	//HORA COMPLETA
	IF 	LA_IHM.HORARIO_ATUAL_SEGUNDO = 59 	AND
		LA_IHM.HORARIO_ATUAL_MINUTO  = 59	THEN
		LA_IHM.bit_HORARIO_HORA_COMPLETO	:=	TRUE;
	ELSE
		LA_IHM.bit_HORARIO_HORA_COMPLETO	:=	FALSE;
	END_IF
	
	//DIA COMPLETO
	IF 	LA_IHM.HORARIO_ATUAL_SEGUNDO = 57 	AND
		LA_IHM.HORARIO_ATUAL_MINUTO  = 59	AND
		LA_IHM.HORARIO_ATUAL_HORA	  = 5	OR
		teste_dia						 	THEN
		LA_IHM.bit_HORARIO_DIA_COMPLETO	:=	TRUE;
	ELSE
		LA_IHM.bit_HORARIO_DIA_COMPLETO	:=	FALSE;
	END_IF
	
	//DIA REAL COMPLETO
	IF 	LA_IHM.HORARIO_ATUAL_SEGUNDO = 58 	AND
		LA_IHM.HORARIO_ATUAL_MINUTO  = 59	AND
		LA_IHM.HORARIO_ATUAL_HORA	  = 23	THEN
		LA_IHM.bit_HORARIO_DIA_COMPLETO_REAL	:=	TRUE;
	ELSE
		LA_IHM.bit_HORARIO_DIA_COMPLETO_REAL	:=	FALSE;
	END_IF

//TIMER RETENTIVOS TURNO MAQUINA RODANDO
pvar.RTON_tmr_MAQUINA_RODANDO_T1(T_IN:= LA_IHM.turno_A AND LA_GERAL.bit_STATUS_RODANDO, T_PT:= T#999999999MS);
pvar.RTON_tmr_MAQUINA_RODANDO_T2(T_IN:= LA_IHM.turno_B AND LA_GERAL.bit_STATUS_RODANDO, T_PT:= T#999999999MS);
pvar.RTON_tmr_MAQUINA_RODANDO_T3(T_IN:= LA_IHM.turno_C AND LA_GERAL.bit_STATUS_RODANDO, T_PT:= T#999999999MS);

//TIMER RETENTIVOS TURNO MAQUINA PARADA
pvar.RTON_tmr_MAQUINA_PARADA_T1(T_IN:= LA_IHM.turno_A AND LA_GERAL.bit_STATUS_PARADA, T_PT:= T#999999999MS);
pvar.RTON_tmr_MAQUINA_PARADA_T2(T_IN:= LA_IHM.turno_B AND LA_GERAL.bit_STATUS_PARADA, T_PT:= T#999999999MS);
pvar.RTON_tmr_MAQUINA_PARADA_T3(T_IN:= LA_IHM.turno_C AND LA_GERAL.bit_STATUS_PARADA, T_PT:= T#999999999MS);

//TIMER RETENTIVOS TURNO MAQUINA OCIOSA
pvar.RTON_tmr_MAQUINA_OCIOSA_T1(T_IN:= LA_IHM.turno_A AND LA_GERAL.bit_STATUS_OCIOSA, T_PT:= T#999999999MS);
pvar.RTON_tmr_MAQUINA_OCIOSA_T2(T_IN:= LA_IHM.turno_B AND LA_GERAL.bit_STATUS_OCIOSA, T_PT:= T#999999999MS);
pvar.RTON_tmr_MAQUINA_OCIOSA_T3(T_IN:= LA_IHM.turno_C AND LA_GERAL.bit_STATUS_OCIOSA, T_PT:= T#999999999MS);

//================================================================================================================================================================================
//================================================================================================================================================================================

//--------//--------//-------//------CONTADORES------//--------------//-----------//-----------//------------//


//CONTAGEM PILHAS PESADAS OK TURNO A
pvar.cont_PILHAS_COMPLETADAS_TURNO_1(
	CU:= GVL_PESAGEM.bit_PESAGEM_ATUAL AND (LA_GERAL.bit_STATUS_RODANDO OR LA_GERAL.bit_STATUS_OCIOSA) AND LA_IHM.turno_A);
	
//CONTAGEM PILHAS PESADAS OK TURNO B
pvar.cont_PILHAS_COMPLETADAS_TURNO_2(
	CU:= GVL_PESAGEM.bit_PESAGEM_ATUAL AND (LA_GERAL.bit_STATUS_RODANDO OR LA_GERAL.bit_STATUS_OCIOSA) AND LA_IHM.turno_B);
	
//CONTAGEM PILHAS PESADAS OK TURNO C
pvar.cont_PILHAS_COMPLETADAS_TURNO_3(
	CU:= GVL_PESAGEM.bit_PESAGEM_ATUAL AND (LA_GERAL.bit_STATUS_RODANDO OR LA_GERAL.bit_STATUS_OCIOSA) AND LA_IHM.turno_C);

//CONTAGEM PILHAS REJEITADAS TURNO A
pvar.cont_PILHAS_REJEITADAS_TURNO_1(
	CU:= GVL_PESAGEM.bit_PESAGEM_ERRO AND (LA_GERAL.bit_STATUS_RODANDO OR LA_GERAL.bit_STATUS_OCIOSA) AND LA_IHM.turno_A);
	
//CONTAGEM PILHAS REJEITADAS TURNO B
pvar.cont_PILHAS_REJEITADAS_TURNO_2(
	CU:= GVL_PESAGEM.bit_PESAGEM_ERRO AND (LA_GERAL.bit_STATUS_RODANDO OR LA_GERAL.bit_STATUS_OCIOSA) AND LA_IHM.turno_B);
	
//CONTAGEM PILHAS REJEITADAS TURNO C
pvar.cont_PILHAS_REJEITADAS_TURNO_3(
	CU:= GVL_PESAGEM.bit_PESAGEM_ERRO AND (LA_GERAL.bit_STATUS_RODANDO OR LA_GERAL.bit_STATUS_OCIOSA) AND LA_IHM.turno_C);
	
//CONTAGEM PILHAS TOTAL TURNO A
pvar.cont_PILHAS_TOTAL_TURNO_1(
	CU:= (GVL_PESAGEM.bit_PESAGEM_ATUAL OR GVL_PESAGEM.bit_PESAGEM_ERRO) AND (LA_GERAL.bit_STATUS_RODANDO OR LA_GERAL.bit_STATUS_OCIOSA OR teste) AND LA_IHM.turno_A);
	
//CONTAGEM PILHAS TOTAL TURNO B
pvar.cont_PILHAS_TOTAL_TURNO_2(
	CU:= (GVL_PESAGEM.bit_PESAGEM_ATUAL OR GVL_PESAGEM.bit_PESAGEM_ERRO) AND (LA_GERAL.bit_STATUS_RODANDO OR LA_GERAL.bit_STATUS_OCIOSA) AND LA_IHM.turno_B);
	
//CONTAGEM PILHAS TOTAL TURNO C
pvar.cont_PILHAS_TOTAL_TURNO_3(
	CU:= (GVL_PESAGEM.bit_PESAGEM_ATUAL OR GVL_PESAGEM.bit_PESAGEM_ERRO) AND (LA_GERAL.bit_STATUS_RODANDO OR LA_GERAL.bit_STATUS_OCIOSA) AND LA_IHM.turno_C);
	
//--------//--------//-------//------EFICIENCIA------//--------------//-----------//-----------//------------//
//garante que não haverá erros de divisão por 0. A eficiencia só é contada a partir de quando a contagem POR TEMPO começou
	
//PORCENTAGEM DE PILHAS COMPLETADAS TURNO 1
IF PVAR.ihm_PILHAS_TOTAL_TURNO_ARRAY.PRIMEIRO[0] > 0 THEN
	LA_IHM.num_PORCENTAGEM_COMPLETADAS_T1	:=	(DINT_TO_REAL(PVAR.ihm_PILHAS_COMPLETADAS_TURNO_ARRAY.PRIMEIRO[0]) / DINT_TO_REAL(PVAR.ihm_PILHAS_TOTAL_TURNO_ARRAY.PRIMEIRO[0])) * 100;
END_IF

//PORCENTAGEM DE PILHAS COMPLETADAS TURNO 2
IF PVAR.ihm_PILHAS_TOTAL_TURNO_ARRAY.SEGUNDO[0] > 0 THEN
	LA_IHM.num_PORCENTAGEM_COMPLETADAS_T2	:=	(DINT_TO_REAL(PVAR.ihm_PILHAS_COMPLETADAS_TURNO_ARRAY.SEGUNDO[0]) / DINT_TO_REAL(PVAR.ihm_PILHAS_TOTAL_TURNO_ARRAY.SEGUNDO[0])) * 100;
END_IF

//PORCENTAGEM DE PILHAS COMPLETADAS TURNO 3
IF PVAR.ihm_PILHAS_TOTAL_TURNO_ARRAY.TERCEIRO[0] > 0 THEN
	LA_IHM.num_PORCENTAGEM_COMPLETADAS_T3	:=	(DINT_TO_REAL(PVAR.ihm_PILHAS_COMPLETADAS_TURNO_ARRAY.TERCEIRO[0]) / DINT_TO_REAL(PVAR.ihm_PILHAS_TOTAL_TURNO_ARRAY.TERCEIRO[0])) * 100;
END_IF


//PORCENTAGEM DE PILHAS REJEITADAS TURNO 1
IF PVAR.ihm_PILHAS_TOTAL_TURNO_ARRAY.PRIMEIRO[0] > 0 THEN
	LA_IHM.num_PORCENTAGEM_REJEITADAS_T1	:=	100 - LA_IHM.num_PORCENTAGEM_COMPLETADAS_T1;
END_IF

//PORCENTAGEM DE PILHAS REJEITADAS TURNO 2
IF PVAR.ihm_PILHAS_TOTAL_TURNO_ARRAY.SEGUNDO[0] > 0 THEN
	LA_IHM.num_PORCENTAGEM_REJEITADAS_T2	:=	100 - LA_IHM.num_PORCENTAGEM_COMPLETADAS_T2;
END_IF

//PORCENTAGEM DE PILHAS REJEITADAS TURNO 3
IF PVAR.ihm_PILHAS_TOTAL_TURNO_ARRAY.TERCEIRO[0] > 0 THEN
	LA_IHM.num_PORCENTAGEM_REJEITADAS_T3	:=	100 - LA_IHM.num_PORCENTAGEM_COMPLETADAS_T3;
END_IF


//================================================================================================================================================================================
//================================================================================================================================================================================
//RESET DE VARIÁVEIS NA TROCA DE TURNO

	IF tmr_TURNO_TROCADO.Q THEN
		pvar.RTON_tmr_MAQUINA_RODANDO_T1.Timer_reset	:=	TRUE;
		pvar.RTON_tmr_MAQUINA_RODANDO_T2.Timer_reset	:=	TRUE;
		pvar.RTON_tmr_MAQUINA_RODANDO_T3.Timer_reset	:=	TRUE;
		
		pvar.RTON_tmr_MAQUINA_PARADA_T1.Timer_reset	:=	TRUE;
		pvar.RTON_tmr_MAQUINA_PARADA_T2.Timer_reset	:=	TRUE;
		pvar.RTON_tmr_MAQUINA_PARADA_T3.Timer_reset	:=	TRUE;
		
		pvar.RTON_tmr_MAQUINA_OCIOSA_T1.Timer_reset	:=	TRUE;
		pvar.RTON_tmr_MAQUINA_OCIOSA_T2.Timer_reset	:=	TRUE;
		pvar.RTON_tmr_MAQUINA_OCIOSA_T3.Timer_reset	:=	TRUE;
		
		PVAR.cont_PILHAS_COMPLETADAS_TURNO_1.RESET	:=	TRUE;
		PVAR.cont_PILHAS_COMPLETADAS_TURNO_2.RESET	:=	TRUE;
		PVAR.cont_PILHAS_COMPLETADAS_TURNO_3.RESET	:=	TRUE;
		
		PVAR.cont_PILHAS_REJEITADAS_TURNO_1.RESET	:=	TRUE;
		PVAR.cont_PILHAS_REJEITADAS_TURNO_2.RESET	:=	TRUE;
		PVAR.cont_PILHAS_REJEITADAS_TURNO_3.RESET	:=	TRUE;
		
		PVAR.cont_PILHAS_TOTAL_TURNO_1.RESET		:=	TRUE;
		PVAR.cont_PILHAS_TOTAL_TURNO_2.RESET		:=	TRUE;
		PVAR.cont_PILHAS_TOTAL_TURNO_3.RESET		:=	TRUE;
		
		LA_GERAL.bit_TURNO_TROCADO				:= FALSE;
	ELSE
		pvar.RTON_tmr_MAQUINA_RODANDO_T1.Timer_reset	:=	FALSE;
		pvar.RTON_tmr_MAQUINA_RODANDO_T2.Timer_reset	:=	FALSE;
		pvar.RTON_tmr_MAQUINA_RODANDO_T3.Timer_reset	:=	FALSE;
		
		pvar.RTON_tmr_MAQUINA_PARADA_T1.Timer_reset	:=	FALSE;
		pvar.RTON_tmr_MAQUINA_PARADA_T2.Timer_reset	:=	FALSE;
		pvar.RTON_tmr_MAQUINA_PARADA_T3.Timer_reset	:=	FALSE;
		
		pvar.RTON_tmr_MAQUINA_OCIOSA_T1.Timer_reset	:=	FALSE;
		pvar.RTON_tmr_MAQUINA_OCIOSA_T2.Timer_reset	:=	FALSE;
		pvar.RTON_tmr_MAQUINA_OCIOSA_T3.Timer_reset	:=	FALSE;
		
		PVAR.cont_PILHAS_COMPLETADAS_TURNO_1.RESET	:=	FALSE;
		PVAR.cont_PILHAS_COMPLETADAS_TURNO_2.RESET	:=	FALSE;
		PVAR.cont_PILHAS_COMPLETADAS_TURNO_3.RESET	:=	FALSE;
		
		PVAR.cont_PILHAS_REJEITADAS_TURNO_1.RESET	:=	FALSE;
		PVAR.cont_PILHAS_REJEITADAS_TURNO_2.RESET	:=	FALSE;
		PVAR.cont_PILHAS_REJEITADAS_TURNO_3.RESET	:=	FALSE;
		
		PVAR.cont_PILHAS_TOTAL_TURNO_1.RESET		:=	FALSE;
		PVAR.cont_PILHAS_TOTAL_TURNO_2.RESET		:=	FALSE;
		PVAR.cont_PILHAS_TOTAL_TURNO_3.RESET		:=	FALSE;
		
	END_IF
	
//RESETAR MANUALMENTE CONTADORES DO TURNO A
	IF LA_IHM.bit_CONTADORES_RESET	AND LA_IHM.turno_A THEN
		pvar.RTON_tmr_MAQUINA_RODANDO_T1.Timer_reset	:=	TRUE;
		pvar.RTON_tmr_MAQUINA_PARADA_T1.Timer_reset		:=	TRUE;
		pvar.RTON_tmr_MAQUINA_OCIOSA_T1.Timer_reset		:=	TRUE;
		PVAR.cont_PILHAS_COMPLETADAS_TURNO_1.RESET		:=	TRUE;
		PVAR.cont_PILHAS_REJEITADAS_TURNO_1.RESET		:=	TRUE;
		PVAR.cont_PILHAS_TOTAL_TURNO_1.RESET			:=	TRUE;
	END_IF
	
//RESETAR MANUALMENTE CONTADORES DO TURNO B
	IF LA_IHM.bit_CONTADORES_RESET	AND LA_IHM.turno_B THEN
		pvar.RTON_tmr_MAQUINA_RODANDO_T2.Timer_reset	:=	TRUE;
		pvar.RTON_tmr_MAQUINA_PARADA_T2.Timer_reset		:=	TRUE;
		pvar.RTON_tmr_MAQUINA_OCIOSA_T2.Timer_reset		:=	TRUE;
		PVAR.cont_PILHAS_COMPLETADAS_TURNO_2.RESET		:=	TRUE;
		PVAR.cont_PILHAS_REJEITADAS_TURNO_2.RESET		:=	TRUE;
		PVAR.cont_PILHAS_TOTAL_TURNO_2.RESET			:=	TRUE;
	END_IF
	
//RESETAR MANUALMENTE CONTADORES DO TURNO C
	IF LA_IHM.bit_CONTADORES_RESET	AND LA_IHM.turno_C THEN
		pvar.RTON_tmr_MAQUINA_RODANDO_T3.Timer_reset	:=	TRUE;
		pvar.RTON_tmr_MAQUINA_PARADA_T3.Timer_reset		:=	TRUE;
		pvar.RTON_tmr_MAQUINA_OCIOSA_T3.Timer_reset		:=	TRUE;
		PVAR.cont_PILHAS_COMPLETADAS_TURNO_3.RESET		:=	TRUE;
		PVAR.cont_PILHAS_REJEITADAS_TURNO_3.RESET		:=	TRUE;
		PVAR.cont_PILHAS_TOTAL_TURNO_3.RESET			:=	TRUE;
	END_IF


//RESETAR CONTADORES DOS TURNOS 05:59:55
	IF 	(LA_IHM.HORARIO_ATUAL_HORA 	 = 5	AND
		LA_IHM.HORARIO_ATUAL_MINUTO = 59		AND
		LA_IHM.HORARIO_ATUAL_SEGUNDO = 55)		OR
		teste_reset_cont_turnoa					THEN
			LA_GERAL.bit_TURNO_TROCADO	:= TRUE;
	END_IF

tmr_TURNO_TROCADO		(IN := LA_GERAL.bit_TURNO_TROCADO,  PT := T#4S);


//LIMITE DE HORÁRIOS DOS TURNOS
LIM_HORA_TURNO1(IN:= LA_IHM.HORARIO_ATUAL_HORA, HIGH:= 13, LOW:= 6);
LIM_HORA_TURNO2(IN:= LA_IHM.HORARIO_ATUAL_HORA, HIGH:= 21, LOW:= 14);
LIM_HORA_TURNO3(IN:= LA_IHM.HORARIO_ATUAL_HORA, HIGH:= 5, LOW:= 22);

E06_HISTORICO();
E07_HISTORICO_ESPELHAMENTO();

END_PROGRAM

// LADO_A/05 - LA_IHM/E06_HISTORICO
PROGRAM E06_HISTORICO
VAR
	HORARIO_ATUAL_DIA_ANTERIOR	: DINT;
END_VAR

	IF LA_IHM.bit_HORARIO_DIA_COMPLETO_REAL THEN
		LA_IHM.info_DIA_ANTERIOR := LA_IHM.HORARIO_ATUAL_DIA;
		LA_IHM.info_MES_ANTERIOR := LA_IHM.HORARIO_ATUAL_MES;
	END_IF
	
//================================================================================================================================================================================
//================================================================================================================================================================================
//ARMAZENAMENTO DE DADOS DE PRODUÇÃO DE TURNO

	//ARMAZENAMENTO DE DADOS DE PRODUÇÃO TURNO A
	IF LA_IHM.turno_A	THEN
		
		PVAR.IHM_DIA_TURNO_ARRAY.PRIMEIRO[0] := LA_IHM.HORARIO_ATUAL_DIA;
		PVAR.IHM_MES_TURNO_ARRAY.PRIMEIRO[0] := LA_IHM.HORARIO_ATUAL_MES;
		
		PVAR.IHM_TEMPO_RODANDO_ARRAY.PRIMEIRO[0] := TIME_TO_DINT(pvar.RTON_tmr_MAQUINA_RODANDO_T1.RTON_ET);
		PVAR.IHM_TEMPO_PARADO_ARRAY.PRIMEIRO[0]  := TIME_TO_DINT(pvar.RTON_tmr_MAQUINA_PARADA_T1.RTON_ET);
		PVAR.IHM_TEMPO_OCIOSO_ARRAY.PRIMEIRO[0]  := TIME_TO_DINT(pvar.RTON_tmr_MAQUINA_OCIOSA_T1.RTON_ET);
	
		PVAR.ihm_PILHAS_COMPLETADAS_TURNO_ARRAY.PRIMEIRO[0]		:=	pvar.cont_PILHAS_COMPLETADAS_TURNO_1.CV;
		PVAR.ihm_PILHAS_REJEITADAS_TURNO_ARRAY.PRIMEIRO[0]		:=	pvar.cont_PILHAS_REJEITADAS_TURNO_1.CV;
		PVAR.ihm_PILHAS_TOTAL_TURNO_ARRAY.PRIMEIRO[0]			:=	pvar.cont_PILHAS_TOTAL_TURNO_1.CV;
		
		PVAR.ihm_PILHAS_COMPLETADAS_PORCENTAGEM_TURNO_ARRAY.PRIMEIRO[0]	:=	REAL_TO_DINT(LA_IHM.num_PORCENTAGEM_COMPLETADAS_T1);
		PVAR.ihm_PILHAS_REJEITADAS_PORCENTAGEM_TURNO_ARRAY.PRIMEIRO[0]	:=	REAL_TO_DINT(LA_IHM.num_PORCENTAGEM_REJEITADAS_T1);
	END_IF
	
	//ARMAZENAMENTO DE DADOS DE PRODUÇÃO TURNO B
	IF LA_IHM.turno_B	THEN
		
		PVAR.IHM_DIA_TURNO_ARRAY.SEGUNDO[0] := LA_IHM.HORARIO_ATUAL_DIA;
		PVAR.IHM_MES_TURNO_ARRAY.SEGUNDO[0] := LA_IHM.HORARIO_ATUAL_MES;
		
		PVAR.IHM_TEMPO_RODANDO_ARRAY.SEGUNDO[0] := TIME_TO_DINT(pvar.RTON_tmr_MAQUINA_RODANDO_T2.RTON_ET);
		PVAR.IHM_TEMPO_PARADO_ARRAY.SEGUNDO[0]  := TIME_TO_DINT(pvar.RTON_tmr_MAQUINA_PARADA_T2.RTON_ET);
		PVAR.IHM_TEMPO_OCIOSO_ARRAY.SEGUNDO[0]  := TIME_TO_DINT(pvar.RTON_tmr_MAQUINA_OCIOSA_T2.RTON_ET);
		
		PVAR.ihm_PILHAS_COMPLETADAS_TURNO_ARRAY.SEGUNDO[0]		:=	pvar.cont_PILHAS_COMPLETADAS_TURNO_2.CV;
		PVAR.ihm_PILHAS_REJEITADAS_TURNO_ARRAY.SEGUNDO[0]		:=	pvar.cont_PILHAS_REJEITADAS_TURNO_2.CV;
		PVAR.ihm_PILHAS_TOTAL_TURNO_ARRAY.SEGUNDO[0]			:=	pvar.cont_PILHAS_TOTAL_TURNO_2.CV;
		
		PVAR.ihm_PILHAS_COMPLETADAS_PORCENTAGEM_TURNO_ARRAY.SEGUNDO[0]	:=	REAL_TO_DINT(LA_IHM.num_PORCENTAGEM_COMPLETADAS_T2);
		PVAR.ihm_PILHAS_REJEITADAS_PORCENTAGEM_TURNO_ARRAY.SEGUNDO[0]	:=	REAL_TO_DINT(LA_IHM.num_PORCENTAGEM_REJEITADAS_T2);
	END_IF
	
	//ARMAZENAMENTO DE DADOS DE PRODUÇÃO TURNO C
	IF LA_IHM.turno_C	THEN
	
	IF LA_IHM.HORARIO_ATUAL_HORA <= 5 THEN
		PVAR.IHM_DIA_TURNO_ARRAY.TERCEIRO[0] := LA_IHM.HORARIO_ATUAL_DIA - 1;
		PVAR.IHM_MES_TURNO_ARRAY.TERCEIRO[0] := LA_IHM.HORARIO_ATUAL_MES;
	ELSE
		PVAR.IHM_DIA_TURNO_ARRAY.TERCEIRO[0] := LA_IHM.HORARIO_ATUAL_DIA;
		PVAR.IHM_MES_TURNO_ARRAY.TERCEIRO[0] := LA_IHM.HORARIO_ATUAL_MES;
	END_IF
		
		PVAR.IHM_TEMPO_RODANDO_ARRAY.TERCEIRO[0] := TIME_TO_DINT(pvar.RTON_tmr_MAQUINA_RODANDO_T3.RTON_ET);
		PVAR.IHM_TEMPO_PARADO_ARRAY.TERCEIRO[0]  := TIME_TO_DINT(pvar.RTON_tmr_MAQUINA_PARADA_T3.RTON_ET);
		PVAR.IHM_TEMPO_OCIOSO_ARRAY.TERCEIRO[0]  := TIME_TO_DINT(pvar.RTON_tmr_MAQUINA_OCIOSA_T3.RTON_ET);
		
		PVAR.ihm_PILHAS_COMPLETADAS_TURNO_ARRAY.TERCEIRO[0]		:=	pvar.cont_PILHAS_COMPLETADAS_TURNO_3.CV;
		PVAR.ihm_PILHAS_REJEITADAS_TURNO_ARRAY.TERCEIRO[0]		:=	pvar.cont_PILHAS_REJEITADAS_TURNO_3.CV;
		PVAR.ihm_PILHAS_TOTAL_TURNO_ARRAY.TERCEIRO[0]			:=	pvar.cont_PILHAS_TOTAL_TURNO_3.CV;
		
		PVAR.ihm_PILHAS_COMPLETADAS_PORCENTAGEM_TURNO_ARRAY.TERCEIRO[0]	:=	REAL_TO_DINT(LA_IHM.num_PORCENTAGEM_COMPLETADAS_T3);
		PVAR.ihm_PILHAS_REJEITADAS_PORCENTAGEM_TURNO_ARRAY.TERCEIRO[0]	:=	REAL_TO_DINT(LA_IHM.num_PORCENTAGEM_REJEITADAS_T3);
	END_IF
	
	
//================================================================================================================================================================================
//================================================================================================================================================================================
//SHIFT NO ARMAZENAMENTO DE DADOS DE PRODUÇÃO DE TURNO

//---------------//---------------DIA COMPLETO PRIMEIRO---------------//---------------//---------------//---------------//---------------//---------------//---------------//---------------//---------------//---------------//---------------//---------------//
	LA_IHM.COP_ihm_DIA_TURNO(Source:= ADR(PVAR.IHM_DIA_TURNO_ARRAY.PRIMEIRO[0]) , Dest:= ADR(PVAR.IHM_DIA_TURNO_ARRAY_AUX.PRIMEIRO[0]), Length:= 10, Trigger:= LA_IHM.bit_HORARIO_DIA_COMPLETO);
	LA_IHM.COP_ihm_DIA_TURNO_AUX(Source:= ADR(PVAR.IHM_DIA_TURNO_ARRAY_AUX.PRIMEIRO[0]) , Dest:= ADR(PVAR.IHM_DIA_TURNO_ARRAY.PRIMEIRO[1]), Length:= 9, Trigger:= LA_IHM.bit_HORARIO_DIA_COMPLETO);
	
	LA_IHM.COP_ihm_MES_TURNO(Source:= ADR(PVAR.IHM_MES_TURNO_ARRAY.PRIMEIRO[0]) , Dest:= ADR(PVAR.IHM_MES_TURNO_ARRAY_AUX.PRIMEIRO[0]), Length:= 10, Trigger:= LA_IHM.bit_HORARIO_DIA_COMPLETO);
	LA_IHM.COP_ihm_MES_TURNO_AUX(Source:= ADR(PVAR.IHM_MES_TURNO_ARRAY_AUX.PRIMEIRO[0]) , Dest:= ADR(PVAR.IHM_MES_TURNO_ARRAY.PRIMEIRO[1]), Length:= 9, Trigger:= LA_IHM.bit_HORARIO_DIA_COMPLETO);
	
	LA_IHM.COP_ihm_RODANDO_TURNO(Source:= ADR(PVAR.IHM_TEMPO_RODANDO_ARRAY.PRIMEIRO[0]) , Dest:= ADR(PVAR.IHM_TEMPO_RODANDO_ARRAY_AUX.PRIMEIRO[0]), Length:= 10, Trigger:= LA_IHM.bit_HORARIO_DIA_COMPLETO);
	LA_IHM.COP_ihm_RODANDO_TURNO_AUX(Source:= ADR(PVAR.IHM_TEMPO_RODANDO_ARRAY_AUX.PRIMEIRO[0]) , Dest:= ADR(PVAR.IHM_TEMPO_RODANDO_ARRAY.PRIMEIRO[1]), Length:= 9, Trigger:= LA_IHM.bit_HORARIO_DIA_COMPLETO);
	
	LA_IHM.COP_ihm_PARADO_TURNO(Source:= ADR(PVAR.IHM_TEMPO_PARADO_ARRAY.PRIMEIRO[0]) , Dest:= ADR(PVAR.IHM_TEMPO_PARADO_ARRAY_AUX.PRIMEIRO[0]), Length:= 10, Trigger:= LA_IHM.bit_HORARIO_DIA_COMPLETO);
	LA_IHM.COP_ihm_PARADO_TURNO_AUX(Source:= ADR(PVAR.IHM_TEMPO_PARADO_ARRAY_AUX.PRIMEIRO[0]) , Dest:= ADR(PVAR.IHM_TEMPO_PARADO_ARRAY.PRIMEIRO[1]), Length:= 9, Trigger:= LA_IHM.bit_HORARIO_DIA_COMPLETO);
	
	LA_IHM.COP_ihm_OCIOSO_TURNO(Source:= ADR(PVAR.IHM_TEMPO_OCIOSO_ARRAY.PRIMEIRO[0]) , Dest:= ADR(PVAR.IHM_TEMPO_OCIOSO_ARRAY_AUX.PRIMEIRO[0]), Length:= 10, Trigger:= LA_IHM.bit_HORARIO_DIA_COMPLETO);
	LA_IHM.COP_ihm_OCIOSO_TURNO_AUX(Source:= ADR(PVAR.IHM_TEMPO_OCIOSO_ARRAY_AUX.PRIMEIRO[0]) , Dest:= ADR(PVAR.IHM_TEMPO_OCIOSO_ARRAY.PRIMEIRO[1]), Length:= 9, Trigger:= LA_IHM.bit_HORARIO_DIA_COMPLETO);
		
	LA_IHM.COP_ihm_PILHAS_COMPLETADAS_TURNO(Source:= ADR(PVAR.ihm_PILHAS_COMPLETADAS_TURNO_ARRAY.PRIMEIRO[0]) , Dest:= ADR(PVAR.ihm_PILHAS_COMPLETADAS_TURNO_ARRAY_AUX.PRIMEIRO[0]), Length:= 10, Trigger:= LA_IHM.bit_HORARIO_DIA_COMPLETO);
	LA_IHM.COP_ihm_PILHAS_COMPLETADAS_TURNO_AUX(Source:= ADR(PVAR.ihm_PILHAS_COMPLETADAS_TURNO_ARRAY_AUX.PRIMEIRO[0]) , Dest:= ADR(PVAR.ihm_PILHAS_COMPLETADAS_TURNO_ARRAY.PRIMEIRO[1]), Length:= 9, Trigger:= LA_IHM.bit_HORARIO_DIA_COMPLETO);
	
	LA_IHM.COP_ihm_PILHAS_REJEITADAS_TURNO(Source:= ADR(PVAR.ihm_PILHAS_REJEITADAS_TURNO_ARRAY.PRIMEIRO[0]) , Dest:= ADR(PVAR.ihm_PILHAS_REJEITADAS_TURNO_ARRAY_AUX.PRIMEIRO[0]), Length:= 10, Trigger:= LA_IHM.bit_HORARIO_DIA_COMPLETO);
	LA_IHM.COP_ihm_PILHAS_REJEITADAS_TURNO_AUX(Source:= ADR(PVAR.ihm_PILHAS_REJEITADAS_TURNO_ARRAY_AUX.PRIMEIRO[0]) , Dest:= ADR(PVAR.ihm_PILHAS_REJEITADAS_TURNO_ARRAY.PRIMEIRO[1]), Length:= 9, Trigger:= LA_IHM.bit_HORARIO_DIA_COMPLETO);
	
	LA_IHM.COP_ihm_PILHAS_TOTAL_TURNO(Source:= ADR(PVAR.ihm_PILHAS_TOTAL_TURNO_ARRAY.PRIMEIRO[0]) , Dest:= ADR(PVAR.ihm_PILHAS_TOTAL_TURNO_ARRAY_AUX.PRIMEIRO[0]), Length:= 10, Trigger:= LA_IHM.bit_HORARIO_DIA_COMPLETO);
	LA_IHM.COP_ihm_PILHAS_TOTAL_TURNO_AUX(Source:= ADR(PVAR.ihm_PILHAS_TOTAL_TURNO_ARRAY_AUX.PRIMEIRO[0]) , Dest:= ADR(PVAR.ihm_PILHAS_TOTAL_TURNO_ARRAY.PRIMEIRO[1]), Length:= 9, Trigger:= LA_IHM.bit_HORARIO_DIA_COMPLETO);
	
	LA_IHM.COP_ihm_PORCENTAGEM_COMPLETADAS(Source:= ADR(PVAR.ihm_PILHAS_COMPLETADAS_PORCENTAGEM_TURNO_ARRAY.PRIMEIRO[0]) , Dest:= ADR(PVAR.ihm_PILHAS_COMPLETADAS_PORCENTAGEM_TURNO_ARRAY_AUX.PRIMEIRO[0]), Length:= 10, Trigger:= LA_IHM.bit_HORARIO_DIA_COMPLETO);
	LA_IHM.COP_ihm_PORCENTAGEM_COMPLETADAS_AUX(Source:= ADR(PVAR.ihm_PILHAS_COMPLETADAS_PORCENTAGEM_TURNO_ARRAY_AUX.PRIMEIRO[0]) , Dest:= ADR(PVAR.ihm_PILHAS_COMPLETADAS_PORCENTAGEM_TURNO_ARRAY.PRIMEIRO[1]), Length:= 9, Trigger:= LA_IHM.bit_HORARIO_DIA_COMPLETO);
	
	LA_IHM.COP_ihm_PORCENTAGEM_REJEITADAS(Source:= ADR(PVAR.ihm_PILHAS_REJEITADAS_PORCENTAGEM_TURNO_ARRAY.PRIMEIRO[0]) , Dest:= ADR(PVAR.ihm_PILHAS_REJEITADAS_PORCENTAGEM_TURNO_ARRAY_AUX.PRIMEIRO[0]), Length:= 10, Trigger:= LA_IHM.bit_HORARIO_DIA_COMPLETO);
	LA_IHM.COP_ihm_PORCENTAGEM_REJEITADAS_AUX(Source:= ADR(PVAR.ihm_PILHAS_REJEITADAS_PORCENTAGEM_TURNO_ARRAY_AUX.PRIMEIRO[0]) , Dest:= ADR(PVAR.ihm_PILHAS_REJEITADAS_PORCENTAGEM_TURNO_ARRAY.PRIMEIRO[1]), Length:= 9, Trigger:= LA_IHM.bit_HORARIO_DIA_COMPLETO);
	
//---------------//---------------//---------------//---------------//---------------//---------------//---------------//---------------//---------------//---------------//---------------//---------------//---------------//---------------//---------------//---------------//	
//---------------//---------------//---------------//---------------//---------------//---------------//---------------//---------------//---------------//---------------//---------------//---------------//---------------//---------------//---------------//---------------//
//---------------//---------------DIA COMPLETO SEGUNDO---------------//---------------//---------------//---------------//---------------//---------------//---------------//---------------//---------------//---------------//---------------//---------------//
	LA_IHM.COP_ihm_DIA_TURNO2(Source:= ADR(PVAR.IHM_DIA_TURNO_ARRAY.SEGUNDO[0]) , Dest:= ADR(PVAR.IHM_DIA_TURNO_ARRAY_AUX.SEGUNDO[0]), Length:= 10, Trigger:= LA_IHM.bit_HORARIO_DIA_COMPLETO);
	LA_IHM.COP_ihm_DIA_TURNO_AUX2(Source:= ADR(PVAR.IHM_DIA_TURNO_ARRAY_AUX.SEGUNDO[0]) , Dest:= ADR(PVAR.IHM_DIA_TURNO_ARRAY.SEGUNDO[1]), Length:= 9, Trigger:= LA_IHM.bit_HORARIO_DIA_COMPLETO);
	
	LA_IHM.COP_ihm_MES_TURNO2(Source:= ADR(PVAR.IHM_MES_TURNO_ARRAY.SEGUNDO[0]) , Dest:= ADR(PVAR.IHM_MES_TURNO_ARRAY_AUX.SEGUNDO[0]), Length:= 10, Trigger:= LA_IHM.bit_HORARIO_DIA_COMPLETO);
	LA_IHM.COP_ihm_MES_TURNO_AUX2(Source:= ADR(PVAR.IHM_MES_TURNO_ARRAY_AUX.SEGUNDO[0]) , Dest:= ADR(PVAR.IHM_MES_TURNO_ARRAY.SEGUNDO[1]), Length:= 9, Trigger:= LA_IHM.bit_HORARIO_DIA_COMPLETO);

	LA_IHM.COP_ihm_RODANDO_TURNO2(Source:= ADR(PVAR.IHM_TEMPO_RODANDO_ARRAY.SEGUNDO[0]) , Dest:= ADR(PVAR.IHM_TEMPO_RODANDO_ARRAY_AUX.SEGUNDO[0]), Length:= 10, Trigger:= LA_IHM.bit_HORARIO_DIA_COMPLETO);
	LA_IHM.COP_ihm_RODANDO_TURNO_AUX2(Source:= ADR(PVAR.IHM_TEMPO_RODANDO_ARRAY_AUX.SEGUNDO[0]) , Dest:= ADR(PVAR.IHM_TEMPO_RODANDO_ARRAY.SEGUNDO[1]), Length:= 9, Trigger:= LA_IHM.bit_HORARIO_DIA_COMPLETO);
	
	LA_IHM.COP_ihm_PARADO_TURNO2(Source:= ADR(PVAR.IHM_TEMPO_PARADO_ARRAY.SEGUNDO[0]) , Dest:= ADR(PVAR.IHM_TEMPO_PARADO_ARRAY_AUX.SEGUNDO[0]), Length:= 10, Trigger:= LA_IHM.bit_HORARIO_DIA_COMPLETO);
	LA_IHM.COP_ihm_PARADO_TURNO_AUX2(Source:= ADR(PVAR.IHM_TEMPO_PARADO_ARRAY_AUX.SEGUNDO[0]) , Dest:= ADR(PVAR.IHM_TEMPO_PARADO_ARRAY.SEGUNDO[1]), Length:= 9, Trigger:= LA_IHM.bit_HORARIO_DIA_COMPLETO);
	
	LA_IHM.COP_ihm_OCIOSO_TURNO2(Source:= ADR(PVAR.IHM_TEMPO_OCIOSO_ARRAY.SEGUNDO[0]) , Dest:= ADR(PVAR.IHM_TEMPO_OCIOSO_ARRAY_AUX.SEGUNDO[0]), Length:= 10, Trigger:= LA_IHM.bit_HORARIO_DIA_COMPLETO);
	LA_IHM.COP_ihm_OCIOSO_TURNO_AUX2(Source:= ADR(PVAR.IHM_TEMPO_OCIOSO_ARRAY_AUX.SEGUNDO[0]) , Dest:= ADR(PVAR.IHM_TEMPO_OCIOSO_ARRAY.SEGUNDO[1]), Length:= 9, Trigger:= LA_IHM.bit_HORARIO_DIA_COMPLETO);
	
	LA_IHM.COP_ihm_PILHAS_COMPLETADAS_TURNO2(Source:= ADR(PVAR.ihm_PILHAS_COMPLETADAS_TURNO_ARRAY.SEGUNDO[0]) , Dest:= ADR(PVAR.ihm_PILHAS_COMPLETADAS_TURNO_ARRAY_AUX.SEGUNDO[0]), Length:= 10, Trigger:= LA_IHM.bit_HORARIO_DIA_COMPLETO);
	LA_IHM.COP_ihm_PILHAS_COMPLETADAS_TURNO_AUX2(Source:= ADR(PVAR.ihm_PILHAS_COMPLETADAS_TURNO_ARRAY_AUX.SEGUNDO[0]) , Dest:= ADR(PVAR.ihm_PILHAS_COMPLETADAS_TURNO_ARRAY.SEGUNDO[1]), Length:= 9, Trigger:= LA_IHM.bit_HORARIO_DIA_COMPLETO);
	
	LA_IHM.COP_ihm_PILHAS_REJEITADAS_TURNO2(Source:= ADR(PVAR.ihm_PILHAS_REJEITADAS_TURNO_ARRAY.SEGUNDO[0]) , Dest:= ADR(PVAR.ihm_PILHAS_REJEITADAS_TURNO_ARRAY_AUX.SEGUNDO[0]), Length:= 10, Trigger:= LA_IHM.bit_HORARIO_DIA_COMPLETO);
	LA_IHM.COP_ihm_PILHAS_REJEITADAS_TURNO_AUX2(Source:= ADR(PVAR.ihm_PILHAS_REJEITADAS_TURNO_ARRAY_AUX.SEGUNDO[0]) , Dest:= ADR(PVAR.ihm_PILHAS_REJEITADAS_TURNO_ARRAY.SEGUNDO[1]), Length:= 9, Trigger:= LA_IHM.bit_HORARIO_DIA_COMPLETO);
	
	LA_IHM.COP_ihm_PILHAS_TOTAL_TURNO2(Source:= ADR(PVAR.ihm_PILHAS_TOTAL_TURNO_ARRAY.SEGUNDO[0]) , Dest:= ADR(PVAR.ihm_PILHAS_TOTAL_TURNO_ARRAY_AUX.SEGUNDO[0]), Length:= 10, Trigger:= LA_IHM.bit_HORARIO_DIA_COMPLETO);
	LA_IHM.COP_ihm_PILHAS_TOTAL_TURNO_AUX2(Source:= ADR(PVAR.ihm_PILHAS_TOTAL_TURNO_ARRAY_AUX.SEGUNDO[0]) , Dest:= ADR(PVAR.ihm_PILHAS_TOTAL_TURNO_ARRAY.SEGUNDO[1]), Length:= 9, Trigger:= LA_IHM.bit_HORARIO_DIA_COMPLETO);
	
	LA_IHM.COP_ihm_PORCENTAGEM_COMPLETADAS2(Source:= ADR(PVAR.ihm_PILHAS_COMPLETADAS_PORCENTAGEM_TURNO_ARRAY.SEGUNDO[0]) , Dest:= ADR(PVAR.ihm_PILHAS_COMPLETADAS_PORCENTAGEM_TURNO_ARRAY_AUX.SEGUNDO[0]), Length:= 10, Trigger:= LA_IHM.bit_HORARIO_DIA_COMPLETO);
	LA_IHM.COP_ihm_PORCENTAGEM_COMPLETADAS_AUX2(Source:= ADR(PVAR.ihm_PILHAS_COMPLETADAS_PORCENTAGEM_TURNO_ARRAY_AUX.SEGUNDO[0]) , Dest:= ADR(PVAR.ihm_PILHAS_COMPLETADAS_PORCENTAGEM_TURNO_ARRAY.SEGUNDO[1]), Length:= 9, Trigger:= LA_IHM.bit_HORARIO_DIA_COMPLETO);
	
	LA_IHM.COP_ihm_PORCENTAGEM_REJEITADAS2(Source:= ADR(PVAR.ihm_PILHAS_REJEITADAS_PORCENTAGEM_TURNO_ARRAY.SEGUNDO[0]) , Dest:= ADR(PVAR.ihm_PILHAS_REJEITADAS_PORCENTAGEM_TURNO_ARRAY_AUX.SEGUNDO[0]), Length:= 10, Trigger:= LA_IHM.bit_HORARIO_DIA_COMPLETO);
	LA_IHM.COP_ihm_PORCENTAGEM_REJEITADAS_AUX2(Source:= ADR(PVAR.ihm_PILHAS_REJEITADAS_PORCENTAGEM_TURNO_ARRAY_AUX.SEGUNDO[0]) , Dest:= ADR(PVAR.ihm_PILHAS_REJEITADAS_PORCENTAGEM_TURNO_ARRAY.SEGUNDO[1]), Length:= 9, Trigger:= LA_IHM.bit_HORARIO_DIA_COMPLETO);
//---------------//---------------//---------------//---------------//---------------//---------------//---------------//---------------//---------------//---------------//---------------//---------------//---------------//---------------//---------------//---------------//	
//---------------//---------------//---------------//---------------//---------------//---------------//---------------//---------------//---------------//---------------//---------------//---------------//---------------//---------------//---------------//---------------//
//---------------//---------------DIA COMPLETO TERCEIRO---------------//---------------//---------------//---------------//---------------//---------------//---------------//---------------//---------------//---------------//---------------//---------------//
	LA_IHM.COP_ihm_DIA_TURNO3(Source:= ADR(PVAR.IHM_DIA_TURNO_ARRAY.TERCEIRO[0]) , Dest:= ADR(PVAR.IHM_DIA_TURNO_ARRAY_AUX.TERCEIRO[0]), Length:= 10, Trigger:= LA_IHM.bit_HORARIO_DIA_COMPLETO);
	LA_IHM.COP_ihm_DIA_TURNO_AUX3(Source:= ADR(PVAR.IHM_DIA_TURNO_ARRAY_AUX.TERCEIRO[0]) , Dest:= ADR(PVAR.IHM_DIA_TURNO_ARRAY.TERCEIRO[1]), Length:= 9, Trigger:= LA_IHM.bit_HORARIO_DIA_COMPLETO);
	
	LA_IHM.COP_ihm_MES_TURNO3(Source:= ADR(PVAR.IHM_MES_TURNO_ARRAY.TERCEIRO[0]) , Dest:= ADR(PVAR.IHM_MES_TURNO_ARRAY_AUX.TERCEIRO[0]), Length:= 10, Trigger:= LA_IHM.bit_HORARIO_DIA_COMPLETO);
	LA_IHM.COP_ihm_MES_TURNO_AUX3(Source:= ADR(PVAR.IHM_MES_TURNO_ARRAY_AUX.TERCEIRO[0]) , Dest:= ADR(PVAR.IHM_MES_TURNO_ARRAY.TERCEIRO[1]), Length:= 9, Trigger:= LA_IHM.bit_HORARIO_DIA_COMPLETO);

	LA_IHM.COP_ihm_RODANDO_TURNO3(Source:= ADR(PVAR.IHM_TEMPO_RODANDO_ARRAY.TERCEIRO[0]) , Dest:= ADR(PVAR.IHM_TEMPO_RODANDO_ARRAY_AUX.TERCEIRO[0]), Length:= 10, Trigger:= LA_IHM.bit_HORARIO_DIA_COMPLETO);
	LA_IHM.COP_ihm_RODANDO_TURNO_AUX3(Source:= ADR(PVAR.IHM_TEMPO_RODANDO_ARRAY_AUX.TERCEIRO[0]) , Dest:= ADR(PVAR.IHM_TEMPO_RODANDO_ARRAY.TERCEIRO[1]), Length:= 9, Trigger:= LA_IHM.bit_HORARIO_DIA_COMPLETO);
	
	LA_IHM.COP_ihm_PARADO_TURNO3(Source:= ADR(PVAR.IHM_TEMPO_PARADO_ARRAY.TERCEIRO[0]) , Dest:= ADR(PVAR.IHM_TEMPO_PARADO_ARRAY_AUX.TERCEIRO[0]), Length:= 10, Trigger:= LA_IHM.bit_HORARIO_DIA_COMPLETO);
	LA_IHM.COP_ihm_PARADO_TURNO_AUX3(Source:= ADR(PVAR.IHM_TEMPO_PARADO_ARRAY_AUX.TERCEIRO[0]) , Dest:= ADR(PVAR.IHM_TEMPO_PARADO_ARRAY.TERCEIRO[1]), Length:= 9, Trigger:= LA_IHM.bit_HORARIO_DIA_COMPLETO);
	
	LA_IHM.COP_ihm_OCIOSO_TURNO3(Source:= ADR(PVAR.IHM_TEMPO_OCIOSO_ARRAY.TERCEIRO[0]) , Dest:= ADR(PVAR.IHM_TEMPO_OCIOSO_ARRAY_AUX.TERCEIRO[0]), Length:= 10, Trigger:= LA_IHM.bit_HORARIO_DIA_COMPLETO);
	LA_IHM.COP_ihm_OCIOSO_TURNO_AUX3(Source:= ADR(PVAR.IHM_TEMPO_OCIOSO_ARRAY_AUX.TERCEIRO[0]) , Dest:= ADR(PVAR.IHM_TEMPO_OCIOSO_ARRAY.TERCEIRO[1]), Length:= 9, Trigger:= LA_IHM.bit_HORARIO_DIA_COMPLETO);
	
	LA_IHM.COP_ihm_PILHAS_COMPLETADAS_TURNO3(Source:= ADR(PVAR.ihm_PILHAS_COMPLETADAS_TURNO_ARRAY.TERCEIRO[0]) , Dest:= ADR(PVAR.ihm_PILHAS_COMPLETADAS_TURNO_ARRAY_AUX.TERCEIRO[0]), Length:= 10, Trigger:= LA_IHM.bit_HORARIO_DIA_COMPLETO);
	LA_IHM.COP_ihm_PILHAS_COMPLETADAS_TURNO_AUX3(Source:= ADR(PVAR.ihm_PILHAS_COMPLETADAS_TURNO_ARRAY_AUX.TERCEIRO[0]) , Dest:= ADR(PVAR.ihm_PILHAS_COMPLETADAS_TURNO_ARRAY.TERCEIRO[1]), Length:= 9, Trigger:= LA_IHM.bit_HORARIO_DIA_COMPLETO);
	
	LA_IHM.COP_ihm_PILHAS_REJEITADAS_TURNO3(Source:= ADR(PVAR.ihm_PILHAS_REJEITADAS_TURNO_ARRAY.TERCEIRO[0]) , Dest:= ADR(PVAR.ihm_PILHAS_REJEITADAS_TURNO_ARRAY_AUX.TERCEIRO[0]), Length:= 10, Trigger:= LA_IHM.bit_HORARIO_DIA_COMPLETO);
	LA_IHM.COP_ihm_PILHAS_REJEITADAS_TURNO_AUX3(Source:= ADR(PVAR.ihm_PILHAS_REJEITADAS_TURNO_ARRAY_AUX.TERCEIRO[0]) , Dest:= ADR(PVAR.ihm_PILHAS_REJEITADAS_TURNO_ARRAY.TERCEIRO[1]), Length:= 9, Trigger:= LA_IHM.bit_HORARIO_DIA_COMPLETO);
	
	LA_IHM.COP_ihm_PILHAS_TOTAL_TURNO3(Source:= ADR(PVAR.ihm_PILHAS_TOTAL_TURNO_ARRAY.TERCEIRO[0]) , Dest:= ADR(PVAR.ihm_PILHAS_TOTAL_TURNO_ARRAY_AUX.TERCEIRO[0]), Length:= 10, Trigger:= LA_IHM.bit_HORARIO_DIA_COMPLETO);
	LA_IHM.COP_ihm_PILHAS_TOTAL_TURNO_AUX3(Source:= ADR(PVAR.ihm_PILHAS_TOTAL_TURNO_ARRAY_AUX.TERCEIRO[0]) , Dest:= ADR(PVAR.ihm_PILHAS_TOTAL_TURNO_ARRAY.TERCEIRO[1]), Length:= 9, Trigger:= LA_IHM.bit_HORARIO_DIA_COMPLETO);
	
	LA_IHM.COP_ihm_PORCENTAGEM_COMPLETADAS3(Source:= ADR(PVAR.ihm_PILHAS_COMPLETADAS_PORCENTAGEM_TURNO_ARRAY.TERCEIRO[0]) , Dest:= ADR(PVAR.ihm_PILHAS_COMPLETADAS_PORCENTAGEM_TURNO_ARRAY_AUX.TERCEIRO[0]), Length:= 10, Trigger:= LA_IHM.bit_HORARIO_DIA_COMPLETO);
	LA_IHM.COP_ihm_PORCENTAGEM_COMPLETADAS_AUX3(Source:= ADR(PVAR.ihm_PILHAS_COMPLETADAS_PORCENTAGEM_TURNO_ARRAY_AUX.TERCEIRO[0]) , Dest:= ADR(PVAR.ihm_PILHAS_COMPLETADAS_PORCENTAGEM_TURNO_ARRAY.TERCEIRO[1]), Length:= 9, Trigger:= LA_IHM.bit_HORARIO_DIA_COMPLETO);
	
	LA_IHM.COP_ihm_PORCENTAGEM_REJEITADAS3(Source:= ADR(PVAR.ihm_PILHAS_REJEITADAS_PORCENTAGEM_TURNO_ARRAY.TERCEIRO[0]) , Dest:= ADR(PVAR.ihm_PILHAS_REJEITADAS_PORCENTAGEM_TURNO_ARRAY_AUX.TERCEIRO[0]), Length:= 10, Trigger:= LA_IHM.bit_HORARIO_DIA_COMPLETO);
	LA_IHM.COP_ihm_PORCENTAGEM_REJEITADAS_AUX3(Source:= ADR(PVAR.ihm_PILHAS_REJEITADAS_PORCENTAGEM_TURNO_ARRAY_AUX.TERCEIRO[0]) , Dest:= ADR(PVAR.ihm_PILHAS_REJEITADAS_PORCENTAGEM_TURNO_ARRAY.TERCEIRO[1]), Length:= 9, Trigger:= LA_IHM.bit_HORARIO_DIA_COMPLETO);

	
LA_IHM.ONS_DIA_COMPLETO_1(CLK := LA_IHM.bit_HORARIO_DIA_COMPLETO);

END_PROGRAM

// LADO_A/05 - LA_IHM/E07_HISTORICO_ESPELHAMENTO
PROGRAM E07_HISTORICO_ESPELHAMENTO
VAR
	Resultado_Hora_Rodando_Turno1 : DINT;
	Resultado_Hora_Rodando_Turno2 : DINT;
	Resultado_Hora_Rodando_Turno3 : DINT;
	Resultado_Hora_Parada_Turno1  : DINT;
	Resultado_Hora_Parada_Turno2  : DINT;
	Resultado_Hora_Parada_Turno3  : DINT;
	Resultado_Hora_Ociosa_Turno1  : DINT;
	Resultado_Hora_Ociosa_Turno2  : DINT;
	Resultado_Hora_Ociosa_Turno3  : DINT;
	
	Resultado_Minuto_Rodando_Turno1 : DINT;
	Resultado_Minuto_Rodando_Turno2 : DINT;
	Resultado_Minuto_Rodando_Turno3 : DINT;
	Resultado_Minuto_Parada_Turno1  : DINT;
	Resultado_Minuto_Parada_Turno2  : DINT;
	Resultado_Minuto_Parada_Turno3  : DINT;
	Resultado_Minuto_Ociosa_Turno1  : DINT;
	Resultado_Minuto_Ociosa_Turno2  : DINT;
	Resultado_Minuto_Ociosa_Turno3  : DINT;
	
	Resultado_Segundo_Rodando_Turno1 : DINT;
	Resultado_Segundo_Rodando_Turno2 : DINT;
	Resultado_Segundo_Rodando_Turno3 : DINT;
	Resultado_Segundo_Parada_Turno1  : DINT;
	Resultado_Segundo_Parada_Turno2  : DINT;
	Resultado_Segundo_Parada_Turno3  : DINT;
	Resultado_Segundo_Ociosa_Turno1  : DINT;
	Resultado_Segundo_Ociosa_Turno2  : DINT;
	Resultado_Segundo_Ociosa_Turno3  : DINT;
	
	Constante_Hora				  : DINT := 3600000;
	Constante_minuto			  : DINT :=	60000;
	Constante_segundo			  : DINT :=	1000;
	
	In_Minutos_Rodando_T1		  : DINT;
	In_Minutos_Rodando_T2		  : DINT;
	In_Minutos_Rodando_T3		  : DINT;
	In_Minutos_Parado_T1		  : DINT;
	In_Minutos_Parado_T2		  : DINT;
	In_Minutos_Parado_T3		  : DINT;
	In_Minutos_Ocioso_T1		  : DINT;
	In_Minutos_Ocioso_T2		  : DINT;
	In_Minutos_Ocioso_T3		  : DINT;
	
	In_Segundos_Rodando_T1		  : DINT;
	In_Segundos_Rodando_T2		  : DINT;
	In_Segundos_Rodando_T3		  : DINT;
	In_Segundos_Parado_T1		  : DINT;
	In_Segundos_Parado_T2		  : DINT;
	In_Segundos_Parado_T3		  : DINT;
	In_Segundos_Ocioso_T1		  : DINT;
	In_Segundos_Ocioso_T2		  : DINT;
	In_Segundos_Ocioso_T3		  : DINT;

	
END_VAR

//================================================================================================================================================================================
//================================================================================================================================================================================
//SELEÇÃO DE DADOS NO INDEX

//SELEÇÃO DE DADOS DO TURNO 1
	IF LA_IHM.ihm_HIST_INDEX_TURNO1[0]	THEN
			LA_GERAL.int_HIST_INDEX_TURNO1	:= 0;
	END_IF
	
	IF LA_IHM.ihm_HIST_INDEX_TURNO1[1]	THEN
			LA_GERAL.int_HIST_INDEX_TURNO1	:= 1;
	END_IF
	
	IF LA_IHM.ihm_HIST_INDEX_TURNO1[2]	THEN
			LA_GERAL.int_HIST_INDEX_TURNO1	:= 2;
	END_IF
	
	IF LA_IHM.ihm_HIST_INDEX_TURNO1[3]	THEN
			LA_GERAL.int_HIST_INDEX_TURNO1	:= 3;
	END_IF
	
	IF LA_IHM.ihm_HIST_INDEX_TURNO1[4]	THEN
			LA_GERAL.int_HIST_INDEX_TURNO1	:= 4;
	END_IF
	
	IF LA_IHM.ihm_HIST_INDEX_TURNO1[5]	THEN
			LA_GERAL.int_HIST_INDEX_TURNO1	:= 5;
	END_IF
	
	IF LA_IHM.ihm_HIST_INDEX_TURNO1[6]	THEN
			LA_GERAL.int_HIST_INDEX_TURNO1	:= 6;
	END_IF
	
	IF LA_IHM.ihm_HIST_INDEX_TURNO1[7]	THEN
			LA_GERAL.int_HIST_INDEX_TURNO1	:= 7;
	END_IF
	
	IF LA_IHM.ihm_HIST_INDEX_TURNO1[8]	THEN
			LA_GERAL.int_HIST_INDEX_TURNO1	:= 8;
	END_IF
	
	IF LA_IHM.ihm_HIST_INDEX_TURNO1[9]	THEN
			LA_GERAL.int_HIST_INDEX_TURNO1	:= 9;
	END_IF
	
//---------------//------------------------------------------//--------------------------------//---------------//------------------------------------------//--------------------------------
//---------------//------------------------------------------//--------------------------------//---------------//------------------------------------------//--------------------------------	
//SELEÇÃO DE DADOS DO TURNO 2
	IF LA_IHM.ihm_HIST_INDEX_TURNO2[0]	THEN
			LA_GERAL.int_HIST_INDEX_TURNO2	:= 0;
	END_IF
	
	IF LA_IHM.ihm_HIST_INDEX_TURNO2[1]	THEN
			LA_GERAL.int_HIST_INDEX_TURNO2	:= 1;
	END_IF
	
	IF LA_IHM.ihm_HIST_INDEX_TURNO2[2]	THEN
			LA_GERAL.int_HIST_INDEX_TURNO2	:= 2;
	END_IF
	
	IF LA_IHM.ihm_HIST_INDEX_TURNO2[3]	THEN
			LA_GERAL.int_HIST_INDEX_TURNO2	:= 3;
	END_IF
	
	IF LA_IHM.ihm_HIST_INDEX_TURNO2[4]	THEN
			LA_GERAL.int_HIST_INDEX_TURNO2	:= 4;
	END_IF
	
	IF LA_IHM.ihm_HIST_INDEX_TURNO2[5]	THEN
			LA_GERAL.int_HIST_INDEX_TURNO2	:= 5;
	END_IF
	
	IF LA_IHM.ihm_HIST_INDEX_TURNO2[6]	THEN
			LA_GERAL.int_HIST_INDEX_TURNO2	:= 6;
	END_IF
	
	IF LA_IHM.ihm_HIST_INDEX_TURNO2[7]	THEN
			LA_GERAL.int_HIST_INDEX_TURNO2	:= 7;
	END_IF
	
	IF LA_IHM.ihm_HIST_INDEX_TURNO2[8]	THEN
			LA_GERAL.int_HIST_INDEX_TURNO2	:= 8;
	END_IF
	
	IF LA_IHM.ihm_HIST_INDEX_TURNO2[9]	THEN
			LA_GERAL.int_HIST_INDEX_TURNO2	:= 9;
	END_IF
	
	
//---------------//------------------------------------------//--------------------------------//---------------//------------------------------------------//--------------------------------
//---------------//------------------------------------------//--------------------------------//---------------//------------------------------------------//--------------------------------	
//SELEÇÃO DE DADOS DO TURNO 3
	IF 	LA_IHM.ihm_HIST_INDEX_TURNO3[0] THEN
			LA_GERAL.int_HIST_INDEX_TURNO3	:= 0;
	END_IF
	
	IF LA_IHM.ihm_HIST_INDEX_TURNO3[1]	THEN
			LA_GERAL.int_HIST_INDEX_TURNO3	:= 1;
	END_IF
	
	IF LA_IHM.ihm_HIST_INDEX_TURNO3[2]	THEN
			LA_GERAL.int_HIST_INDEX_TURNO3	:= 2;
	END_IF
	
	IF LA_IHM.ihm_HIST_INDEX_TURNO3[3]	THEN
			LA_GERAL.int_HIST_INDEX_TURNO3	:= 3;
	END_IF
	
	IF LA_IHM.ihm_HIST_INDEX_TURNO3[4]	THEN
			LA_GERAL.int_HIST_INDEX_TURNO3	:= 4;
	END_IF
	
	IF LA_IHM.ihm_HIST_INDEX_TURNO3[5]	THEN
			LA_GERAL.int_HIST_INDEX_TURNO3	:= 5;
	END_IF
	
	IF LA_IHM.ihm_HIST_INDEX_TURNO3[6]	THEN
			LA_GERAL.int_HIST_INDEX_TURNO3	:= 6;
	END_IF
	
	IF LA_IHM.ihm_HIST_INDEX_TURNO3[7]	THEN
			LA_GERAL.int_HIST_INDEX_TURNO3	:= 7;
	END_IF
	
	IF LA_IHM.ihm_HIST_INDEX_TURNO3[8]	THEN
			LA_GERAL.int_HIST_INDEX_TURNO3	:= 8;
	END_IF
	
	IF LA_IHM.ihm_HIST_INDEX_TURNO3[9]	THEN
			LA_GERAL.int_HIST_INDEX_TURNO3	:= 9;
	END_IF
	
//================================================================================================================================================================================
//================================================================================================================================================================================
//ESCREVER DADOS DO INDEX DOS TURNOS

//---------------//---------------INDEX TURNO 1---------------//---------------//---------------//---------------//---------------//---------------//---------------//---------------//---------------//---------------//---------------//---------------//
	LA_IHM.num_PILHAS_COMPLETADAS_T1	:= 	pvar.ihm_PILHAS_COMPLETADAS_TURNO_ARRAY.PRIMEIRO[LA_GERAL.int_HIST_INDEX_TURNO1];
	LA_IHM.num_PILHAS_REJEITADAS_T1	:= 	pvar.ihm_PILHAS_REJEITADAS_TURNO_ARRAY.PRIMEIRO[LA_GERAL.int_HIST_INDEX_TURNO1];
	LA_IHM.num_PILHAS_TOTAL_T1  		:= 	pvar.ihm_PILHAS_TOTAL_TURNO_ARRAY.PRIMEIRO[LA_GERAL.int_HIST_INDEX_TURNO1];
	
	LA_IHM.tmr_MAQUINA_RODANDO_T1 	:= 	pvar.ihm_TEMPO_RODANDO_ARRAY.PRIMEIRO[LA_GERAL.int_HIST_INDEX_TURNO1];
	LA_IHM.tmr_MAQUINA_PARADA_T1 	:= 	pvar.ihm_TEMPO_PARADO_ARRAY.PRIMEIRO[LA_GERAL.int_HIST_INDEX_TURNO1];
	LA_IHM.tmr_MAQUINA_OCIOSA_T1 	:= 	pvar.ihm_TEMPO_OCIOSO_ARRAY.PRIMEIRO[LA_GERAL.int_HIST_INDEX_TURNO1];
	
	LA_IHM.ihm_HIST_PORCENTAGEM_COMPLETADAS_T1  	:= 	pvar.ihm_PILHAS_COMPLETADAS_PORCENTAGEM_TURNO_ARRAY.PRIMEIRO[LA_GERAL.int_HIST_INDEX_TURNO1];
	LA_IHM.ihm_HIST_PORCENTAGEM_REJEITADAS_T1  	:= 	pvar.ihm_PILHAS_REJEITADAS_PORCENTAGEM_TURNO_ARRAY.PRIMEIRO[LA_GERAL.int_HIST_INDEX_TURNO1];
	
	//CONVERSÃO DE HORA / MINUTO / SEGUNDO DE STATUS DA MÁQUINA PARA IHM
	Resultado_Hora_Rodando_Turno1 		:= 	LA_IHM.tmr_MAQUINA_RODANDO_T1 / Constante_Hora;
	In_Minutos_Rodando_T1				:=	LA_IHM.tmr_MAQUINA_RODANDO_T1 MOD Constante_Hora;
	Resultado_Minuto_Rodando_Turno1		:=	In_Minutos_Rodando_T1 / Constante_minuto;
	In_Segundos_Rodando_T1				:=	LA_IHM.tmr_MAQUINA_RODANDO_T1 MOD Constante_minuto;
	Resultado_Segundo_Rodando_Turno1	:=	In_Segundos_Rodando_T1 / Constante_segundo;
	
	Resultado_Hora_Parada_Turno1 		:= 	LA_IHM.tmr_MAQUINA_PARADA_T1 / Constante_Hora;
	In_Minutos_Parado_T1				:=	LA_IHM.tmr_MAQUINA_PARADA_T1 MOD Constante_Hora;
	Resultado_Minuto_Parada_Turno1		:=	In_Minutos_Parado_T1 / Constante_minuto;
	In_Segundos_Parado_T1				:=	LA_IHM.tmr_MAQUINA_PARADA_T1 MOD Constante_minuto;
	Resultado_Segundo_Parada_Turno1		:=	In_Segundos_Parado_T1 / Constante_segundo;
	
	Resultado_Hora_Ociosa_Turno1 		:= 	LA_IHM.tmr_MAQUINA_OCIOSA_T1 / Constante_Hora;
	In_Minutos_Ocioso_T1				:=	LA_IHM.tmr_MAQUINA_OCIOSA_T1 MOD Constante_Hora;
	Resultado_Minuto_Ociosa_Turno1		:=	In_Minutos_Ocioso_T1 / Constante_minuto;
	In_Segundos_Ocioso_T1				:=	LA_IHM.tmr_MAQUINA_OCIOSA_T1 MOD Constante_minuto;
	Resultado_Segundo_Ociosa_Turno1		:=	In_Segundos_Ocioso_T1 / Constante_segundo;
	
	LA_IHM.num_MAQUINA_RODANDO_HORAS_T1 := Resultado_Hora_Rodando_Turno1;
	LA_IHM.num_MAQUINA_PARADA_HORAS_T1 := Resultado_Hora_Parada_Turno1;
	LA_IHM.num_MAQUINA_OCIOSA_HORAS_T1 := Resultado_Hora_Ociosa_Turno1;
	
	LA_IHM.num_MAQUINA_RODANDO_MINUTOS_T1 := Resultado_Minuto_Rodando_Turno1;
	LA_IHM.num_MAQUINA_PARADA_MINUTOS_T1 := Resultado_Minuto_Parada_Turno1;
	LA_IHM.num_MAQUINA_OCIOSA_MINUTOS_T1 := Resultado_Minuto_Ociosa_Turno1;
	
	LA_IHM.num_MAQUINA_RODANDO_SEGUNDOS_T1 := Resultado_Segundo_Rodando_Turno1;
	LA_IHM.num_MAQUINA_PARADA_SEGUNDOS_T1 := Resultado_Segundo_Parada_Turno1;
	LA_IHM.num_MAQUINA_OCIOSA_SEGUNDOS_T1 := Resultado_Segundo_Ociosa_Turno1;

	
//---------------//---------------INDEX TURNO 2---------------//---------------//---------------//---------------//---------------//---------------//---------------//---------------//---------------//---------------//---------------//---------------//
	LA_IHM.num_PILHAS_COMPLETADAS_T2	:= 	pvar.ihm_PILHAS_COMPLETADAS_TURNO_ARRAY.SEGUNDO[LA_GERAL.int_HIST_INDEX_TURNO2];
	LA_IHM.num_PILHAS_REJEITADAS_T2	:= 	pvar.ihm_PILHAS_REJEITADAS_TURNO_ARRAY.SEGUNDO[LA_GERAL.int_HIST_INDEX_TURNO2];
	LA_IHM.num_PILHAS_TOTAL_T2  		:= 	pvar.ihm_PILHAS_TOTAL_TURNO_ARRAY.SEGUNDO[LA_GERAL.int_HIST_INDEX_TURNO2];
	
	LA_IHM.tmr_MAQUINA_RODANDO_T2 	:= 	pvar.ihm_TEMPO_RODANDO_ARRAY.SEGUNDO[LA_GERAL.int_HIST_INDEX_TURNO2];
	LA_IHM.tmr_MAQUINA_PARADA_T2 	:= 	pvar.ihm_TEMPO_PARADO_ARRAY.SEGUNDO[LA_GERAL.int_HIST_INDEX_TURNO2];
	LA_IHM.tmr_MAQUINA_OCIOSA_T2 	:= 	pvar.ihm_TEMPO_OCIOSO_ARRAY.SEGUNDO[LA_GERAL.int_HIST_INDEX_TURNO2];
	
	LA_IHM.ihm_HIST_PORCENTAGEM_COMPLETADAS_T2  	:= 	pvar.ihm_PILHAS_COMPLETADAS_PORCENTAGEM_TURNO_ARRAY.SEGUNDO[LA_GERAL.int_HIST_INDEX_TURNO2];
	LA_IHM.ihm_HIST_PORCENTAGEM_REJEITADAS_T2  	:= 	pvar.ihm_PILHAS_REJEITADAS_PORCENTAGEM_TURNO_ARRAY.SEGUNDO[LA_GERAL.int_HIST_INDEX_TURNO2];
	
	//CONVERSÃO DE HORA / MINUTO / SEGUNDO DE STATUS DA MÁQUINA PARA IHM
	Resultado_Hora_Rodando_Turno2 		:= 	LA_IHM.tmr_MAQUINA_RODANDO_T2 / Constante_Hora;
	In_Minutos_Rodando_T2				:=	LA_IHM.tmr_MAQUINA_RODANDO_T2 MOD Constante_Hora;
	Resultado_Minuto_Rodando_Turno2		:=	In_Minutos_Rodando_T2 / Constante_minuto;
	In_Segundos_Rodando_T2				:=	LA_IHM.tmr_MAQUINA_RODANDO_T2 MOD Constante_minuto;
	Resultado_Segundo_Rodando_Turno2	:=	In_Segundos_Rodando_T2 / Constante_segundo;
	
	Resultado_Hora_Parada_Turno2 		:= 	LA_IHM.tmr_MAQUINA_PARADA_T2 / Constante_Hora;
	In_Minutos_Parado_T2				:=	LA_IHM.tmr_MAQUINA_PARADA_T2 MOD Constante_Hora;
	Resultado_Minuto_Parada_Turno2		:=	In_Minutos_Parado_T2 / Constante_minuto;
	In_Segundos_Parado_T2				:=	LA_IHM.tmr_MAQUINA_PARADA_T2 MOD Constante_minuto;
	Resultado_Segundo_Parada_Turno2		:=	In_Segundos_Parado_T2 / Constante_segundo;
	
	Resultado_Hora_Ociosa_Turno2 		:= 	LA_IHM.tmr_MAQUINA_OCIOSA_T2 / Constante_Hora;
	In_Minutos_Ocioso_T2				:=	LA_IHM.tmr_MAQUINA_OCIOSA_T2 MOD Constante_Hora;
	Resultado_Minuto_Ociosa_Turno2		:=	In_Minutos_Ocioso_T2 / Constante_minuto;
	In_Segundos_Ocioso_T2				:=	LA_IHM.tmr_MAQUINA_OCIOSA_T2 MOD Constante_minuto;
	Resultado_Segundo_Ociosa_Turno2		:=	In_Segundos_Ocioso_T2 / Constante_segundo;

	
	LA_IHM.num_MAQUINA_RODANDO_HORAS_T2 := Resultado_Hora_Rodando_Turno2;
	LA_IHM.num_MAQUINA_PARADA_HORAS_T2 := Resultado_Hora_Parada_Turno2;
	LA_IHM.num_MAQUINA_OCIOSA_HORAS_T2 := Resultado_Hora_Ociosa_Turno2;
	
	LA_IHM.num_MAQUINA_RODANDO_MINUTOS_T2 := Resultado_Minuto_Rodando_Turno2;
	LA_IHM.num_MAQUINA_PARADA_MINUTOS_T2 := Resultado_Minuto_Parada_Turno2;
	LA_IHM.num_MAQUINA_OCIOSA_MINUTOS_T2 := Resultado_Minuto_Ociosa_Turno2;
	
	LA_IHM.num_MAQUINA_RODANDO_SEGUNDOS_T2 := Resultado_Segundo_Rodando_Turno2;
	LA_IHM.num_MAQUINA_PARADA_SEGUNDOS_T2 := Resultado_Segundo_Parada_Turno2;
	LA_IHM.num_MAQUINA_OCIOSA_SEGUNDOS_T2 := Resultado_Segundo_Ociosa_Turno2;

	
	//---------------//---------------INDEX TURNO 3---------------//---------------//---------------//---------------//---------------//---------------//---------------//---------------//---------------//---------------//---------------//---------------//
	LA_IHM.num_PILHAS_COMPLETADAS_T3	:= 	pvar.ihm_PILHAS_COMPLETADAS_TURNO_ARRAY.TERCEIRO[LA_GERAL.int_HIST_INDEX_TURNO3];
	LA_IHM.num_PILHAS_REJEITADAS_T3	:= 	pvar.ihm_PILHAS_REJEITADAS_TURNO_ARRAY.TERCEIRO[LA_GERAL.int_HIST_INDEX_TURNO3];
	LA_IHM.num_PILHAS_TOTAL_T3  		:= 	pvar.ihm_PILHAS_TOTAL_TURNO_ARRAY.TERCEIRO[LA_GERAL.int_HIST_INDEX_TURNO3];
	
	LA_IHM.tmr_MAQUINA_RODANDO_T3 	:= 	pvar.ihm_TEMPO_RODANDO_ARRAY.TERCEIRO[LA_GERAL.int_HIST_INDEX_TURNO3];
	LA_IHM.tmr_MAQUINA_PARADA_T3 	:= 	pvar.ihm_TEMPO_PARADO_ARRAY.TERCEIRO[LA_GERAL.int_HIST_INDEX_TURNO3];
	LA_IHM.tmr_MAQUINA_OCIOSA_T3 	:= 	pvar.ihm_TEMPO_OCIOSO_ARRAY.TERCEIRO[LA_GERAL.int_HIST_INDEX_TURNO3];
	
	LA_IHM.ihm_HIST_PORCENTAGEM_COMPLETADAS_T3  	:= 	pvar.ihm_PILHAS_COMPLETADAS_PORCENTAGEM_TURNO_ARRAY.TERCEIRO[LA_GERAL.int_HIST_INDEX_TURNO2];
	LA_IHM.ihm_HIST_PORCENTAGEM_REJEITADAS_T3  	:= 	pvar.ihm_PILHAS_REJEITADAS_PORCENTAGEM_TURNO_ARRAY.TERCEIRO[LA_GERAL.int_HIST_INDEX_TURNO2];
	
	//CONVERSÃO DE HORA / MINUTO / SEGUNDO DE STATUS DA MÁQUINA PARA IHM
	Resultado_Hora_Rodando_Turno3 		:= 	LA_IHM.tmr_MAQUINA_RODANDO_T3 / Constante_Hora;
	In_Minutos_Rodando_T3				:=	LA_IHM.tmr_MAQUINA_RODANDO_T3 MOD Constante_Hora;
	Resultado_Minuto_Rodando_Turno3		:=	In_Minutos_Rodando_T3 / Constante_minuto;
	In_Segundos_Rodando_T3				:=	LA_IHM.tmr_MAQUINA_RODANDO_T3 MOD Constante_minuto;
	Resultado_Segundo_Rodando_Turno3	:=	In_Segundos_Rodando_T3 / Constante_segundo;
	
	Resultado_Hora_Parada_Turno3 		:= 	LA_IHM.tmr_MAQUINA_PARADA_T3 / Constante_Hora;
	In_Minutos_Parado_T3				:=	LA_IHM.tmr_MAQUINA_PARADA_T3 MOD Constante_Hora;
	Resultado_Minuto_Parada_Turno3		:=	In_Minutos_Parado_T3 / Constante_minuto;
	In_Segundos_Parado_T3				:=	LA_IHM.tmr_MAQUINA_PARADA_T3 MOD Constante_minuto;
	Resultado_Segundo_Parada_Turno3		:=	In_Segundos_Parado_T3 / Constante_segundo;
	
	Resultado_Hora_Ociosa_Turno3 		:= 	LA_IHM.tmr_MAQUINA_OCIOSA_T3 / Constante_Hora;
	In_Minutos_Ocioso_T3				:=	LA_IHM.tmr_MAQUINA_OCIOSA_T3 MOD Constante_Hora;
	Resultado_Minuto_Ociosa_Turno3		:=	In_Minutos_Ocioso_T3 / Constante_minuto;
	In_Segundos_Ocioso_T3				:=	LA_IHM.tmr_MAQUINA_OCIOSA_T3 MOD Constante_minuto;
	Resultado_Segundo_Ociosa_Turno3		:=	In_Segundos_Ocioso_T3 / Constante_segundo;
	
	LA_IHM.num_MAQUINA_RODANDO_HORAS_T3 := Resultado_Hora_Rodando_Turno3;
	LA_IHM.num_MAQUINA_PARADA_HORAS_T3 	:= Resultado_Hora_Parada_Turno3;
	LA_IHM.num_MAQUINA_OCIOSA_HORAS_T3 	:= Resultado_Hora_Ociosa_Turno3;
	
	LA_IHM.num_MAQUINA_RODANDO_MINUTOS_T3 := Resultado_Minuto_Rodando_Turno3;
	LA_IHM.num_MAQUINA_PARADA_MINUTOS_T3 	:= Resultado_Minuto_Parada_Turno3;
	LA_IHM.num_MAQUINA_OCIOSA_MINUTOS_T3 := Resultado_Minuto_Ociosa_Turno3;
	
	LA_IHM.num_MAQUINA_RODANDO_SEGUNDOS_T3 := Resultado_Segundo_Rodando_Turno3;
	LA_IHM.num_MAQUINA_PARADA_SEGUNDOS_T3 := Resultado_Segundo_Parada_Turno3;
	LA_IHM.num_MAQUINA_OCIOSA_SEGUNDOS_T3 := Resultado_Segundo_Ociosa_Turno3;

END_PROGRAM
